Yaskawa INFORM job: R1_W59,61(0,0).JBI

/JOB
//NAME R1_W59,61(0,0)
///FOLDERNAME KRIS-SCIANA
//POS
///NPOS 51,51,0,3,0,0
///TOOL 0
///POSTYPE PULSE
///PULSE
C00000=134415,-715,-4864,-25015,38915,-63413
C00001=113502,8114,43192,26798,43968,-43496
C00002=115630,14888,52648,27203,41243,-43339
C00003=116501,19796,58651,27511,39937,-43351
C00004=117250,23835,63827,27859,38729,-43401
C00005=116459,17865,56800,27447,40081,-43321
C00006=124846,17940,54478,7784,40700,-34045
C00007=125424,19239,56757,7633,39921,-33846
C00008=124253,19371,54731,7961,41326,-34263
C00009=123687,16111,50115,8032,42532,-34411
C00010=122233,8687,39612,8265,45292,-34814
C00011=126161,-17324,-3875,5510,58276,-32288
C00012=137941,4059,13677,718,79048,-46216
C00013=143824,33213,61180,-2695,80182,-57693
C00014=144583,34475,66777,-2587,77412,-57393
C00015=144894,35179,69272,-2544,76248,-57271
C00016=145822,38684,74717,-2397,74726,-56948
C00017=144894,35179,69272,-2544,76248,-57271
C00018=121285,8259,49977,32409,65622,-85655
C00019=121666,7474,49824,32520,65229,-85633
C00020=121151,9880,51545,32428,65555,-85731
C00021=120483,9209,49294,32124,66669,-85644
C00022=122018,5002,33160,30831,72815,-83260
C00023=134158,53958,76682,38239,34179,-24897
C00024=137708,47696,62047,31566,37586,-20771
C00025=134063,25982,44009,42709,43635,-31294
C00026=133982,50047,71636,37367,35128,-24446
C00027=134672,53583,77146,38389,33585,-24905
C00028=122011,28981,48428,46436,51477,-33624
C00029=119605,27506,46763,46738,52879,-34204
C00030=115967,32125,55821,49065,52548,-36550
C00031=118485,34451,59239,49292,50642,-36264
C00032=115423,41017,70943,52033,49745,-38803
C00033=114891,43411,74705,52790,49343,-39446
C00034=113798,45449,78541,53726,49105,-40340
C00035=123524,28907,39088,40151,51076,-28234
C00036=134178,35767,36700,28446,47092,-19134
C00037=143543,32445,26233,33090,88427,-27327
C00038=161050,53810,76540,39832,106879,-39512
C00039=160991,49035,63396,41267,111246,-37738
C00040=155220,20339,35253,49824,102466,-32047
C00041=156950,21555,39558,49933,100203,-32385
C00042=160463,54046,76057,39663,107458,-39537
C00043=160676,56960,80197,39521,106547,-39804
C00044=159728,36957,53244,35986,108371,-38729
C00045=158788,19254,34625,20027,98446,-44198
C00046=161065,53727,76445,18583,104001,-45816
C00047=161064,53729,76447,18583,104001,-45817
C00048=161052,53801,76529,18576,103990,-45823
C00049=148287,-6752,-11043,23073,104579,-39820
C00050=134415,-715,-4864,-25015,38915,-63413
BC00000=304677,470241,919133
BC00001=310143,381192,712086
BC00002=310143,381192,712086
BC00003=310143,381192,712086
BC00004=310143,381192,712086
BC00005=310143,381192,712086
BC00006=310143,381192,712086
BC00007=310143,381192,712086
BC00008=310143,381192,712086
BC00009=310143,381192,712086
BC00010=310143,381192,712086
BC00011=310143,381192,712086
BC00012=318680,413372,742266
BC00013=325049,437381,764783
BC00014=325049,437381,764783
BC00015=325049,437381,764783
BC00016=325049,437381,764783
BC00017=325049,437381,764783
BC00018=325049,437381,764779
BC00019=325049,437381,764783
BC00020=325049,437381,764783
BC00021=325049,437381,764783
BC00022=325049,437381,764783
BC00023=345935,445983,759292
BC00024=345977,445988,651758
BC00025=339573,409920,637441
BC00026=339409,438378,637075
BC00027=339409,438378,637075
BC00028=339573,409920,556531
BC00029=339573,409920,556531
BC00030=339573,409920,556531
BC00031=339573,409920,556531
BC00032=339573,409920,556531
BC00033=339573,409920,556531
BC00034=339573,409920,556531
BC00035=359113,424011,538964
BC00036=386365,445714,529170
BC00037=381040,413406,666245
BC00038=390786,379907,741053
BC00039=390828,379912,633518
BC00040=385084,388260,621352
BC00041=385084,388260,621352
BC00042=385004,388377,621184
BC00043=385004,388377,621184
BC00044=398174,388205,551082
BC00045=387556,400319,597186
BC00046=388397,397907,603207
BC00047=390500,391875,618260
BC00048=390458,391870,725795
BC00049=362867,388202,721085
BC00050=304677,549589,919133
///POSTYPE BASE
///RECTAN
///RCONF 0,0,0,0,1,0,0,0,0,0,0,0,0,0,0,0,0,0,0,0,0,0,0,0
P00006=2.006,1.622,-0.565,0.0000,0.0000,0.0000
P00021=0.073,2.058,-0.109,0.0000,0.0000,0.0000
///RCONF 0,0,0,0,0,0,0,0,0,0,0,0,0,0,0,0,0,0,0,0,0,0,0,0
P00023=-2.957,-4.083,2.762,0.0000,0.0000,0.0000
//INST
///DATE 2023/12/07 18:21
///ATTR SC,RW
///GROUP1 RB1,BS1
NOP
'r2_W59,61(0,0)
'Path S1177 (for W883)
SFTOF
MOVJ C00000 BC00000 VJ=50.00
MOVJ C00001 BC00001 VJ=50.00
MOVJ C00002 BC00002 VJ=50.00
MOVL C00003 BC00003 V=60.0
REFP 3 C00004 BC00004
CALL JOB:SEARCH-R1
SET P021 P006
SFTON P021
MOVL C00005 BC00005 V=60.0
MOVL C00006 BC00006 V=60.0
REFP 3 C00007 BC00007
CALL JOB:SEARCH-R1
SET P021 P006
SFTON P021
MOVL C00008 BC00008 V=60.0
MOVL C00009 BC00009 V=100.0
MOVL C00010 BC00010 V=100.0
MOVJ C00011 BC00011 VJ=50.00
'Path S1181 (for W18)
SFTOF
MOVJ C00012 BC00012 VJ=50.00
MOVJ C00013 BC00013 VJ=50.00
MOVJ C00014 BC00014 VJ=50.00
MOVL C00015 BC00015 V=60.0
REFP 3 C00016 BC00016
CALL JOB:SEARCH-R1
SET P023 P006
SFTON P023
MOVL C00017 BC00017 V=60.0
MOVL C00018 BC00018 V=60.0
REFP 3 C00019 BC00019
CALL JOB:SEARCH-R1
SET P023 P006
SFTON P023
MOVL C00020 BC00020 V=60.0
MOVL C00021 BC00021 V=100.0
MOVL C00022 BC00022 V=166.7
'Path W1184
SFTOF
MOVJ C00023 BC00023 VJ=50.00
SFTON P021
MOVJ C00024 BC00024 VJ=50.00
MOVL C00025 BC00025 V=100.0 PL=0
REFP 1 C00026 BC00026
REFP 2 C00027 BC00027
MACRO1 MJ#(0) ARGF10
ARCON
MOVL C00028 BC00028 V=14.2
ARCOF
MOVL C00029 BC00029 V=100.0
MOVL C00030 BC00030 V=100.0
MOVL C00031 BC00031 V=100.0 PL=0
MACRO1 MJ#(0) ARGF10
ARCON
MOVL C00032 BC00032 V=14.2
MOVL C00033 BC00033 V=14.2
MOVL C00034 BC00034 V=14.2
ARCOF
MOVL C00035 BC00035 V=100.0
MOVL C00036 BC00036 V=200.0
SFTOF
'Path W1189
SFTOF
SFTON P023
MOVJ C00037 BC00037 VJ=80.00
MOVJ C00038 BC00038 VJ=80.00
MOVJ C00039 BC00039 VJ=100.00
MOVL C00040 BC00040 V=166.7
MOVL C00041 BC00041 V=100.0 PL=0
REFP 1 C00042 BC00042
REFP 2 C00043 BC00043
MACRO1 MJ#(0) ARGF10
ARCON
MOVL C00044 BC00044 V=13.3
MOVL C00045 BC00045 V=13.3
ARCOF
MOVL C00046 BC00046 V=100.0
MOVL C00047 BC00047 V=200.0
MOVL C00048 BC00048 V=333.3
SFTOF
MOVJ C00049 BC00049 VJ=100.00
MOVJ C00050 BC00050 VJ=100.00
END
